TYPE Position :
	STRUCT
		x, y, theta, e : LREAL; //e = Fehler des Kamerasystems
	END_STRUCT
END_TYPE

(* stored: Version 1.1.0.1, ProductVersion 3.1.4026.13
   DUT Position: Id {2c214e57-e470-4fca-9392-7b725ecf93b5} *)
